SUBAPPLICATION HysteresisParams_AR (* Buendelt MI/DEAD/HYSTERESIS als 3 feste AR-Konstanten (initval_AR) fuer DualHysteresis_AR_AX/_A2X - Werte per Parameter am Aufruf einstellbar *)
  (* Standard: 61499-2; Description: Copyright (c) 2026 Meisterschulen am Ostbahnhof This program and the accompanying materials are made available under the terms of the Eclipse Public License 2.0 which is available at https://www.eclipse.org/legal/epl-2.0/ SPDX-License-Identifier: EPL-2.0 *)
  (* Version 1.0, 2026-09-07, Franz Höpfinger, Meisterschulen am Ostbahnhof, initial API and implementation and/or initial documentation *)
  PACKAGE MyLib::sys;
  (* Documentation:
  MI/DEAD/HYSTERESIS als 3 feste AR-Konstanten gebündelt
   Fasst die drei initval_AR-Instanzen, die DualHysteresis_AR_AX/ _AR_A2X für ihre Parameter-Sockets (MI, DEAD, HYSTERESIS) brauchen, zu einem Baustein zusammen - statt sie in jeder Übung/SubApp einzeln zu wiederholen (wie zuerst in Uebung_234_AX/Uebung_235_AX geschehen).
   Funktionsbeschreibung
    - rMI/rDEAD/rHYSTERESIS sind normale InputVars mit sinnvollen Standardwerten (500.0/20.0/30.0) - am Aufruf per Parameter überschreibbar, genau wie u16ObjId bei den GreenWhiteBackground- Bausteinen.
   - Je ein initval_AR wandelt den jeweiligen Wert in einen festen AR-Plug um, der direkt an DualHysteresis_AR_AX.MI/.DEAD/ .HYSTERESIS (bzw. _AR_A2X) angeschlossen wird.
    Verwendet in Uebung_234_AX (Hardware) und Uebung_235_AX (VT) - identische Parameter, damit beide Übungen direkt vergleichbar bleiben.
  *)
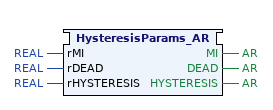
  VAR_INPUT
    rMI : REAL := 500.0; (* Mittelwert/Sollwert *)
    rDEAD : REAL := 20.0; (* Totzone um MI (absolut) *)
    rHYSTERESIS : REAL := 30.0; (* Hysterese zusaetzlich zur Totzone (absolut) *)
  END_VAR
  PLUGS
    MI : adapter::types::unidirectional::AR;
    DEAD : adapter::types::unidirectional::AR;
    HYSTERESIS : adapter::types::unidirectional::AR;
  END_PLUGS
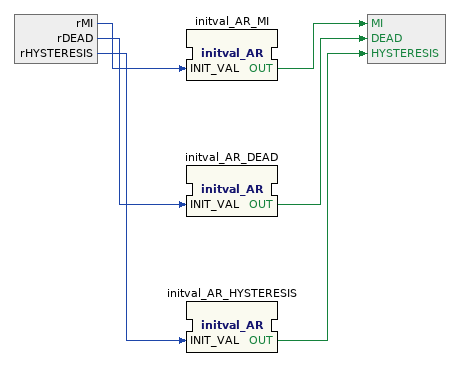
  FBS
    initval_AR_MI : adapter::types::unidirectional::AR::initval::initval_AR;
    initval_AR_DEAD : adapter::types::unidirectional::AR::initval::initval_AR;
    initval_AR_HYSTERESIS : adapter::types::unidirectional::AR::initval::initval_AR;
  END_FBS
  DATA_CONNECTIONS
    rMI TO initval_AR_MI.INIT_VAL;
    rDEAD TO initval_AR_DEAD.INIT_VAL;
    rHYSTERESIS TO initval_AR_HYSTERESIS.INIT_VAL;
  END_CONNECTIONS
  ADAPTER_CONNECTIONS
    initval_AR_MI.OUT TO MI;
    initval_AR_DEAD.OUT TO DEAD;
    initval_AR_HYSTERESIS.OUT TO HYSTERESIS;
  END_CONNECTIONS
END_SUBAPPLICATION
